// TIA Portal V19 export
FUNCTION_BLOCK "FDevice_Contactor_FB"   // FB52, F_LAD
// stored: Access Published
   VAR_INPUT
      FEEDBACK : Bool;
      QBAD_FIO : Bool;
      Estop : Bool;
      Two_Hand_CMD : Bool;   // Safe Motion Command
      Door_SafeStop : Bool;   // Safe Stop from Doors
      CtrlSafe : Bool;   // Movement is Required
      Reset : Bool;
      FeedbackTime : Time := T#200MS;
      StoppingTime : Time := T#2S;   // Movement stopping time
   END_VAR
   VAR_OUTPUT
      OUT : Bool;
      ERROR : Bool;
   END_VAR
   VAR_IN_OUT
      DSI : "udt_DeviceSafetyInterface";   // Device Safety Interface
   END_VAR
   VAR
      DEV : FDBACK;
      T_StopDelay : TOF;
   END_VAR
   VAR_TEMP
      S_ON : Bool;
   END_VAR
BEGIN

REGION Network 1: Safety Enable
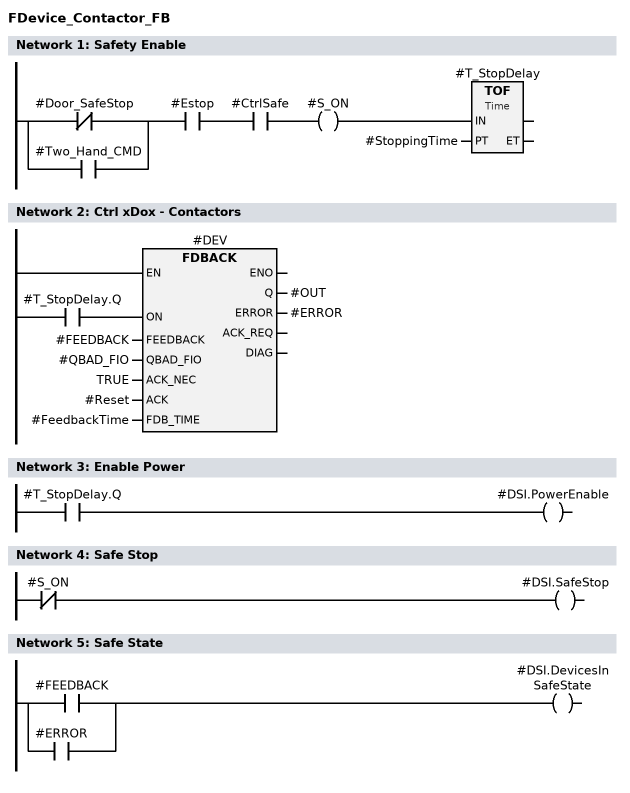
   RUNG wire#powerrail
      I_Contact( #Door_SafeStop )
      wire#w1
      Contact( #Estop )
      Contact( #CtrlSafe )
      Coil( #S_ON )
      { S7_Templates := "[time_type := Time, codedbool_type := DInt]" } #T_StopDelay.TOF(pt := #StoppingTime, et =>)
   END_RUNG
   RUNG wire#powerrail
      Contact( #Two_Hand_CMD )
   END_RUNG wire#w1
   // the same network as SCL:
   #S_ON := (NOT #Door_SafeStop OR #Two_Hand_CMD) AND #Estop AND #CtrlSafe;
   #T_StopDelay.TOF(IN := #S_ON, PT := #StoppingTime);
END_REGION

REGION Network 2: Ctrl xDox - Contactors
   RUNG wire#powerrail
      #DEV.FDBACK(ON := wire#w1, FEEDBACK := #FEEDBACK, QBAD_FIO := #QBAD_FIO, ACK_NEC := TRUE, ACK := #Reset, FDB_TIME := #FeedbackTime, Q => #OUT, ERROR => #ERROR, ACK_REQ =>, DIAG =>)
   END_RUNG
   RUNG wire#powerrail
      Contact( #T_StopDelay.Q )
   END_RUNG wire#w1
   // the same network as SCL:
   #DEV(ON := #T_StopDelay.Q,   // FDBACK
        FEEDBACK := #FEEDBACK,
        QBAD_FIO := #QBAD_FIO,
        ACK_NEC := TRUE,
        ACK := #Reset,
        FDB_TIME := #FeedbackTime,
        Q => #OUT,
        ERROR => #ERROR);
END_REGION

REGION Network 3: Enable Power
   RUNG wire#powerrail
      Contact( #T_StopDelay.Q )
      Coil( #DSI.PowerEnable )
   END_RUNG
   // the same network as SCL:
   #DSI.PowerEnable := #T_StopDelay.Q;
END_REGION

REGION Network 4: Safe Stop
   RUNG wire#powerrail
      I_Contact( #S_ON )
      Coil( #DSI.SafeStop )
   END_RUNG
   // the same network as SCL:
   #DSI.SafeStop := NOT #S_ON;
END_REGION

REGION Network 5: Safe State
   RUNG wire#powerrail
      Contact( #FEEDBACK )
      wire#w1
      Coil( #DSI.DevicesInSafeState )
   END_RUNG
   RUNG wire#powerrail
      Contact( #ERROR )
   END_RUNG wire#w1
   // the same network as SCL:
   #DSI.DevicesInSafeState := #FEEDBACK OR #ERROR;
END_REGION
END_FUNCTION_BLOCK
